// TIA Portal V17 export
// export: Created 2024-08-26T21:10:53.8902487Z, ExportSetting WithDefaults, DisplayName Totally Integrated Automation Portal, DisplayVersion V17 Update 7, DisplayName TIA Portal Openness, DisplayVersion V17 Update 7, DisplayName TIA Portal Version Control Interface, DisplayVersion V17, DisplayName SINAMICS Startdrive Advanced, DisplayVersion V17 SP2, DisplayName SINAMICS Startdrive G110M, G120, G120C, G120D, G120P, G115D, DisplayVersion V17 SP2, DisplayName SINAMICS Startdrive G130, G150, S120, S150, SINAMICS MV, S210, DisplayVersion V17 SP2, DisplayName STEP 7 Professional, DisplayVersion V17 Update 7, DisplayName STEP 7 Safety, DisplayVersion V17 Update 6, DisplayName WinCC Advanced / Unified PC, DisplayVersion V17 Update 7
VAR_GLOBAL   // PLC tag table "clockMemory"
   Clock_Byte AT %MB1 : Byte;
   Clocks_100ms_FP AT %M1.0 : Bool;
   Clocks_200ms_FP AT %M1.1 : Bool;
   Clocks_400ms_FP AT %M1.2 : Bool;
   Clocks_500ms_FP AT %M1.3 : Bool;
   Clocks_800ms_FP AT %M1.4 : Bool;
   Clocks_1s_FP AT %M1.5 : Bool;
   Clocks_1S600ms_FP AT %M1.6 : Bool;
   Clocks_2s_FP AT %M1.7 : Bool;
END_VAR
